Staubli VAL3: onF4Event.pgx

program onF4Event(bool& x_bSave[])
  local bool l_bCheck
  local string l_sMessage
  local frame l_fNewWorld
begin
  // look if the bButton is enable
  if bButton[3]
    //
    if !cycleStatus:bCycle
      if nIndexTool!=0
        call tcp:checkPoint(l_bCheck)
        if l_bCheck
          call tcp:compose(nIndexTool)
          call tcp:getTool(tTool,nIndexTool)
          fFrame=saveData:fFrameItem[saveData:nFrameActive].fFrame
          $jogContext(tTool,fFrame,0)
          logMsg("[KERNEL] INTERFACE:Compose the TCP")
          x_bSave=true
        else
          call language:message(l_sMessage,122)
          popUpMsg(l_sMessage)
        endIf
      endIf
    endIf
  endIf
end
